// TIA Portal V16 export
// export: Created 2022-01-12T14:32:03.2995137Z, ExportSetting WithDefaults, DisplayName Totally Integrated Automation Portal, DisplayVersion V16 Update 4, DisplayName TIA Portal Version Control Interface, DisplayVersion V16 Update 2, DisplayName TIA Portal Openness, DisplayVersion V16 Update 4, DisplayName STEP 7 Professional, DisplayVersion V16 Update 4, DisplayName STEP 7 Safety, DisplayVersion V16, DisplayName WinCC Professional, DisplayVersion V16 Update 4
DATA_BLOCK "Tor2_hmi"   // DB3
{ S7_Optimized_Access := 'TRUE' }
VERSION : 0.1
// stored: AutoNumber true, DBAccessibleFromOPCUA true, IsOnlyStoredInLoadMemory false, IsRetainMemResEnabled false, IsWriteProtectedInAS false, MemoryReserve 100
   VAR
      button { S7_SetPoint := 'True'} : "typKlawiszeProdukcji";
      bPomińŁugowanie { S7_SetPoint := 'True'} : Bool;
      bPomińKwasowanie : Bool;
      bPomińDesynfekcje : Bool;
      bPomińPłukaniePoDezynfekcji : Bool;
   END_VAR
BEGIN
   button.bStart.widoczny := true;
END_DATA_BLOCK
